{attribute 'TcGenerated'}
{attribute 'no-analysis'}
{attribute 'linkalways'}
// This function has been automatically generated from the project information.
VAR_GLOBAL CONSTANT
	{attribute 'const_non_replaced'}
	stLibVersion_CNM_AssertionInterfaces : ST_LibVersion := (iMajor := 0, iMinor := 1, iBuild := 1, iRevision := 0, nFlags := 0, sVersion := '0.1.1.0');
END_VAR

(* stored: Version 1.1.0.1, ProductVersion 3.1.4026.13
   GVL Global_Version: Id {fa4e5a58-0543-4242-9c3d-b8f823118431} *)
